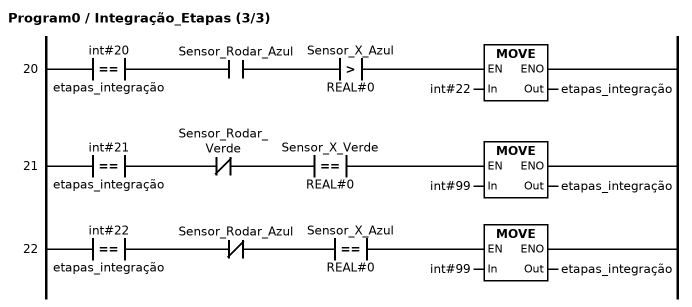
(* [picture p48: Program0 / Integração_Etapas, rungs 20-22] *)
(* Rung 20 *)
IF (int#20 = etapas_integração) AND Sensor_Rodar_Azul AND (Sensor_X_Azul > REAL#0) THEN
    etapas_integração := int#22;
END_IF;
(* Rung 21 *)
IF (int#21 = etapas_integração) AND NOT Sensor_Rodar_Verde AND (Sensor_X_Verde = REAL#0) THEN
    etapas_integração := int#99;
END_IF;
(* Rung 22 *)
IF (int#22 = etapas_integração) AND NOT Sensor_Rodar_Azul AND (Sensor_X_Azul = REAL#0) THEN
    etapas_integração := int#99;
END_IF;

(* Section Integração_Saídas: ladder, written here as Structured Text *)

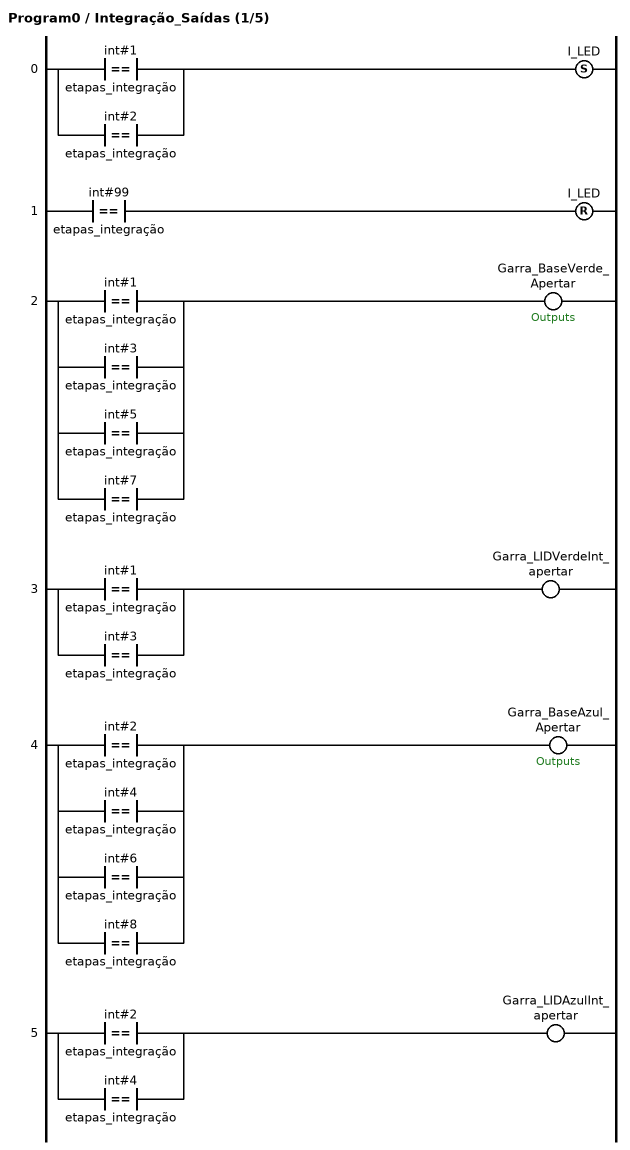
(* Rung 0 *)
IF (int#1 = etapas_integração) OR (int#2 = etapas_integração) THEN I_LED := TRUE; END_IF;
(* Rung 1 *)
IF int#99 = etapas_integração THEN I_LED := FALSE; END_IF;
(* Rung 2 *)
Garra_BaseVerde_Apertar := (int#1 = etapas_integração) OR (int#3 = etapas_integração) OR (int#5 = etapas_integração) OR (int#7 = etapas_integração);
(* Rung 3 *)
Garra_LIDVerdeInt_apertar := (int#1 = etapas_integração) OR (int#3 = etapas_integração);
(* Rung 4 *)
Garra_BaseAzul_Apertar := (int#2 = etapas_integração) OR (int#4 = etapas_integração) OR (int#6 = etapas_integração) OR (int#8 = etapas_integração);
(* Rung 5 *)
Garra_LIDAzulInt_apertar := (int#2 = etapas_integração) OR (int#4 = etapas_integração);

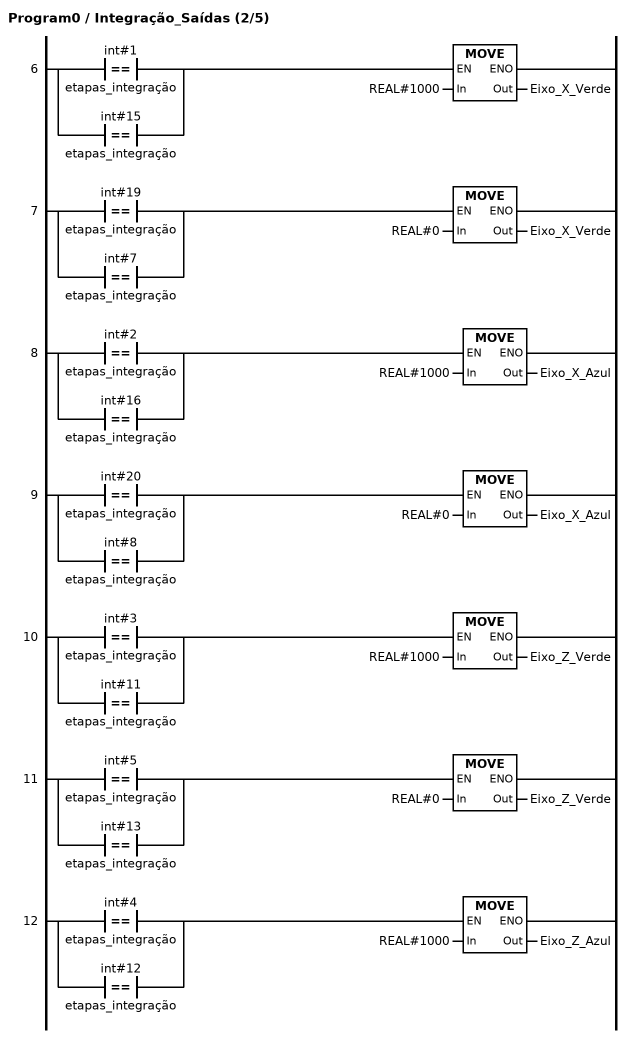
(* Rung 6 *)
IF (int#1 = etapas_integração) OR (int#15 = etapas_integração) THEN Eixo_X_Verde := REAL#1000; END_IF;
(* Rung 7 *)
IF (int#19 = etapas_integração) OR (int#7 = etapas_integração) THEN Eixo_X_Verde := REAL#0; END_IF;
(* Rung 8 *)
IF (int#2 = etapas_integração) OR (int#16 = etapas_integração) THEN Eixo_X_Azul := REAL#1000; END_IF;
(* Rung 9 *)
IF (int#20 = etapas_integração) OR (int#8 = etapas_integração) THEN Eixo_X_Azul := REAL#0; END_IF;
(* Rung 10 *)
IF (int#3 = etapas_integração) OR (int#11 = etapas_integração) THEN Eixo_Z_Verde := REAL#1000; END_IF;
(* Rung 11 *)
IF (int#5 = etapas_integração) OR (int#13 = etapas_integração) THEN Eixo_Z_Verde := REAL#0; END_IF;
(* Rung 12 *)
IF (int#4 = etapas_integração) OR (int#12 = etapas_integração) THEN Eixo_Z_Azul := REAL#1000; END_IF;

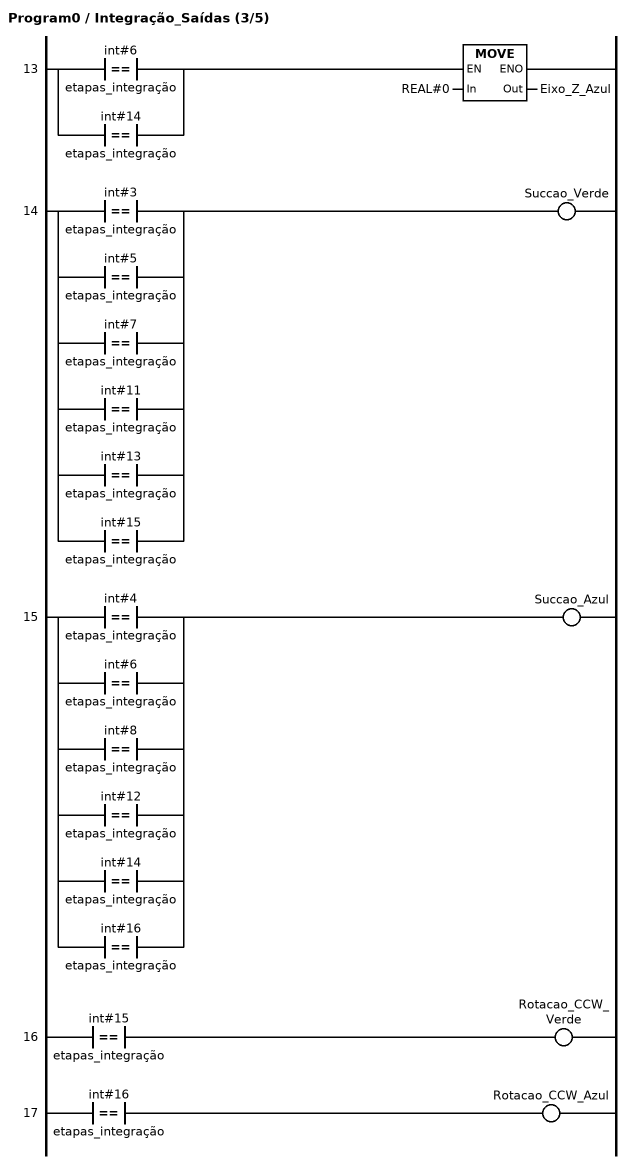
(* Rung 13 *)
IF (int#6 = etapas_integração) OR (int#14 = etapas_integração) THEN Eixo_Z_Azul := REAL#0; END_IF;
(* Rung 14 *)
Succao_Verde := (int#3 = etapas_integração) OR (int#5 = etapas_integração) OR (int#7 = etapas_integração) OR (int#11 = etapas_integração) OR (int#13 = etapas_integração) OR (int#15 = etapas_integração);
(* Rung 15 *)
Succao_Azul := (int#4 = etapas_integração) OR (int#6 = etapas_integração) OR (int#8 = etapas_integração) OR (int#12 = etapas_integração) OR (int#14 = etapas_integração) OR (int#16 = etapas_integração);
(* Rung 16 *)
Rotacao_CCW_Verde := int#15 = etapas_integração;
(* Rung 17 *)
Rotacao_CCW_Azul := int#16 = etapas_integração;

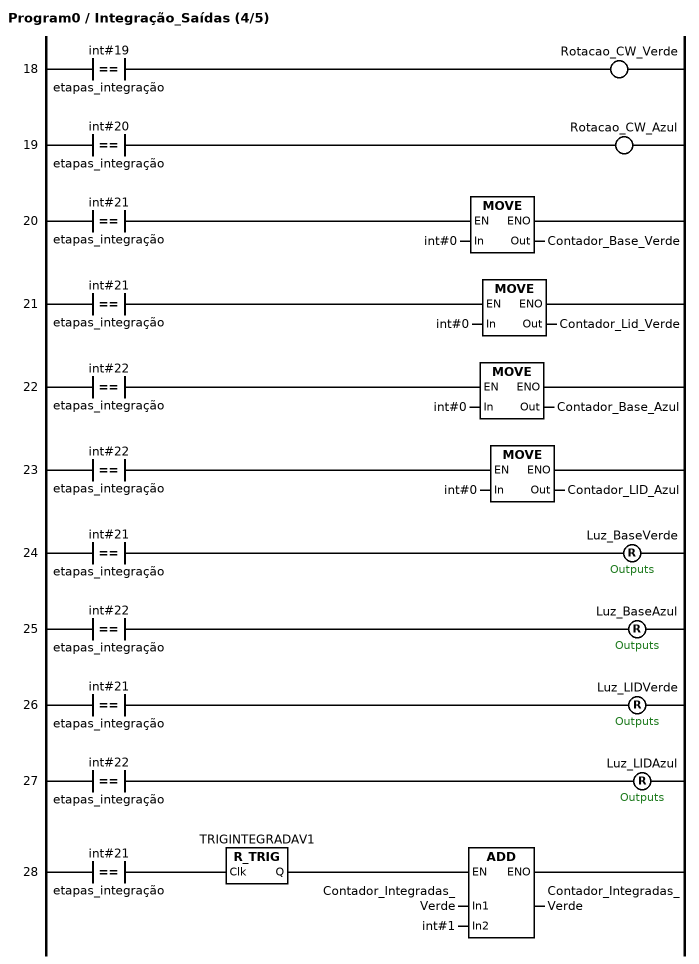
(* Rung 18 *)
Rotacao_CW_Verde := int#19 = etapas_integração;
(* Rung 19 *)
Rotacao_CW_Azul := int#20 = etapas_integração;
(* Rung 20 *)
IF int#21 = etapas_integração THEN Contador_Base_Verde := int#0; END_IF;
(* Rung 21 *)
IF int#21 = etapas_integração THEN Contador_Lid_Verde := int#0; END_IF;
(* Rung 22 *)
IF int#22 = etapas_integração THEN Contador_Base_Azul := int#0; END_IF;
(* Rung 23 *)
IF int#22 = etapas_integração THEN Contador_LID_Azul := int#0; END_IF;
(* Rung 24 *)
IF int#21 = etapas_integração THEN Luz_BaseVerde := FALSE; END_IF;
(* Rung 25 *)
IF int#22 = etapas_integração THEN Luz_BaseAzul := FALSE; END_IF;
(* Rung 26 *)
IF int#21 = etapas_integração THEN Luz_LIDVerde := FALSE; END_IF;
(* Rung 27 *)
IF int#22 = etapas_integração THEN Luz_LIDAzul := FALSE; END_IF;
(* Rung 28 *)
TRIGINTEGRADAV1(Clk := int#21 = etapas_integração);
IF TRIGINTEGRADAV1.Q THEN Contador_Integradas_Verde := Contador_Integradas_Verde + int#1; END_IF;

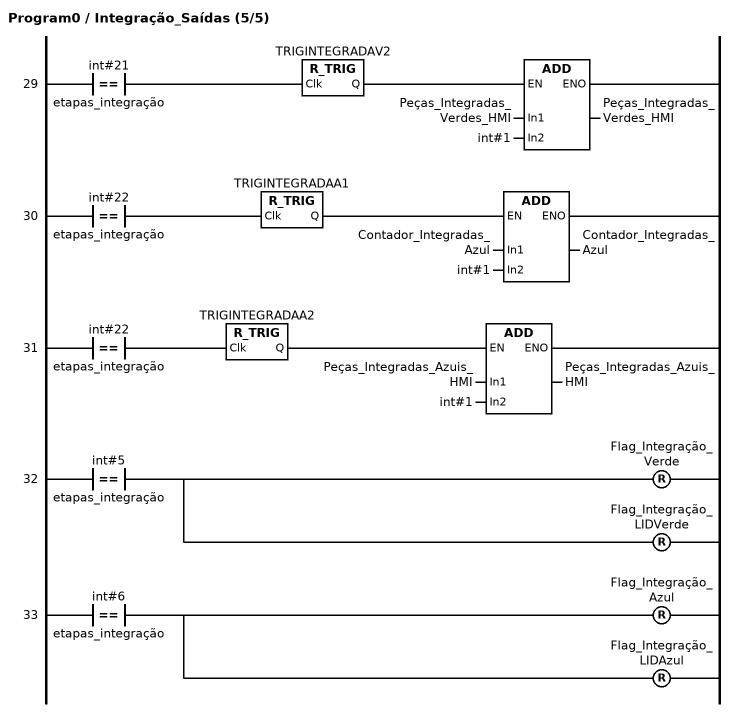
(* Rung 29 *)
TRIGINTEGRADAV2(Clk := int#21 = etapas_integração);
IF TRIGINTEGRADAV2.Q THEN Peças_Integradas_Verdes_HMI := Peças_Integradas_Verdes_HMI + int#1; END_IF;
(* Rung 30 *)
TRIGINTEGRADAA1(Clk := int#22 = etapas_integração);
IF TRIGINTEGRADAA1.Q THEN Contador_Integradas_Azul := Contador_Integradas_Azul + int#1; END_IF;
(* Rung 31 *)
TRIGINTEGRADAA2(Clk := int#22 = etapas_integração);
IF TRIGINTEGRADAA2.Q THEN Peças_Integradas_Azuis_HMI := Peças_Integradas_Azuis_HMI + int#1; END_IF;
(* Rung 32 *)
IF int#5 = etapas_integração THEN
    Flag_Integração_Verde := FALSE;
    Flag_Integração_LIDVerde := FALSE;
END_IF;
(* Rung 33 *)
IF int#6 = etapas_integração THEN
    Flag_Integração_Azul := FALSE;
    Flag_Integração_LIDAzul := FALSE;
END_IF;

(* Section Organização_Etapas: ladder, written here as Structured Text *)

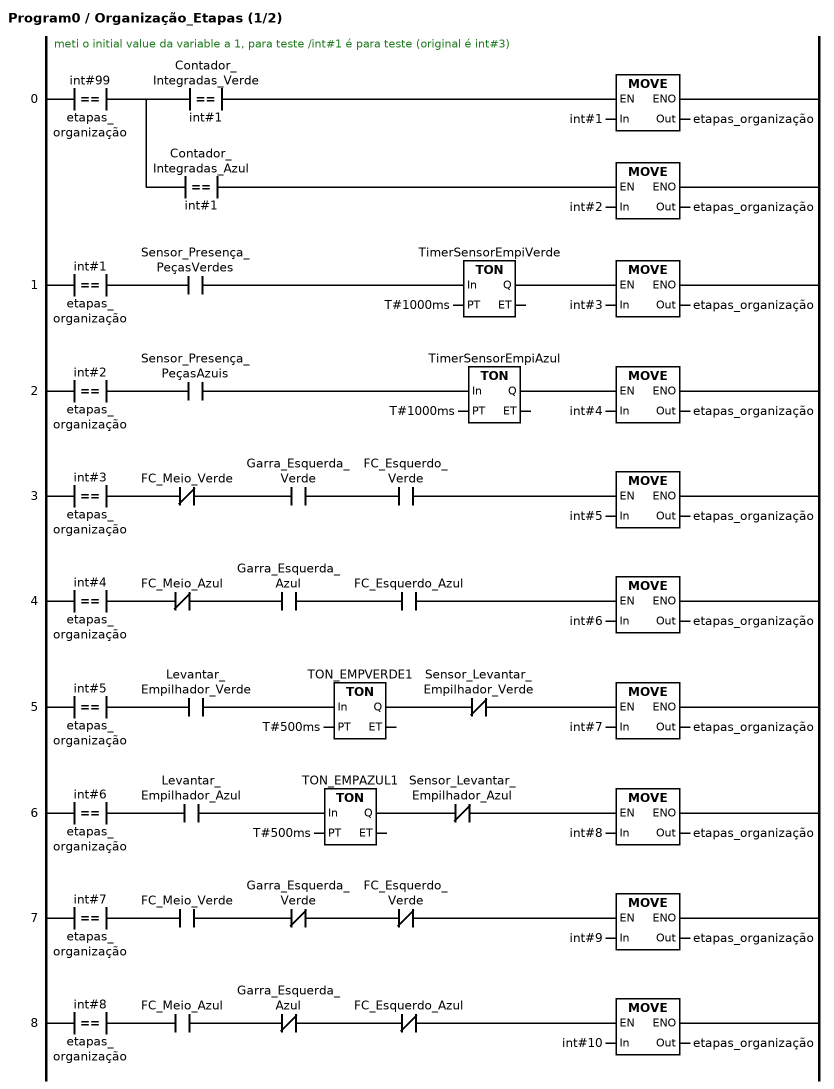
(* Rung 0: meti o initial value da variable a 1, para teste /int#1 é para teste (original é int#3) *)
_p11 := int#99 = etapas_organização;
IF (int#99 = etapas_organização) AND (Contador_Integradas_Verde = int#1) THEN
    etapas_organização := int#1;
END_IF;
IF _p11 AND (Contador_Integradas_Azul = int#1) THEN etapas_organização := int#2; END_IF;
(* Rung 1 *)
TimerSensorEmpiVerde(In := (int#1 = etapas_organização) AND Sensor_Presença_PeçasVerdes, PT := T#1000ms);
IF TimerSensorEmpiVerde.Q THEN etapas_organização := int#3; END_IF;
(* Rung 2 *)
TimerSensorEmpiAzul(In := (int#2 = etapas_organização) AND Sensor_Presença_PeçasAzuis, PT := T#1000ms);
IF TimerSensorEmpiAzul.Q THEN etapas_organização := int#4; END_IF;
(* Rung 3 *)
IF (int#3 = etapas_organização) AND NOT FC_Meio_Verde AND Garra_Esquerda_Verde AND FC_Esquerdo_Verde THEN
    etapas_organização := int#5;
END_IF;
(* Rung 4 *)
IF (int#4 = etapas_organização) AND NOT FC_Meio_Azul AND Garra_Esquerda_Azul AND FC_Esquerdo_Azul THEN
    etapas_organização := int#6;
END_IF;
(* Rung 5 *)
TON_EMPVERDE1(In := (int#5 = etapas_organização) AND Levantar_Empilhador_Verde, PT := T#500ms);
IF TON_EMPVERDE1.Q AND NOT Sensor_Levantar_Empilhador_Verde THEN etapas_organização := int#7; END_IF;
(* Rung 6 *)
TON_EMPAZUL1(In := (int#6 = etapas_organização) AND Levantar_Empilhador_Azul, PT := T#500ms);
IF TON_EMPAZUL1.Q AND NOT Sensor_Levantar_Empilhador_Azul THEN etapas_organização := int#8; END_IF;
(* Rung 7 *)
IF (int#7 = etapas_organização) AND FC_Meio_Verde AND NOT Garra_Esquerda_Verde AND NOT FC_Esquerdo_Verde THEN
    etapas_organização := int#9;
END_IF;
(* Rung 8 *)
IF (int#8 = etapas_organização) AND FC_Meio_Azul AND NOT Garra_Esquerda_Azul AND NOT FC_Esquerdo_Azul THEN
    etapas_organização := int#10;
END_IF;

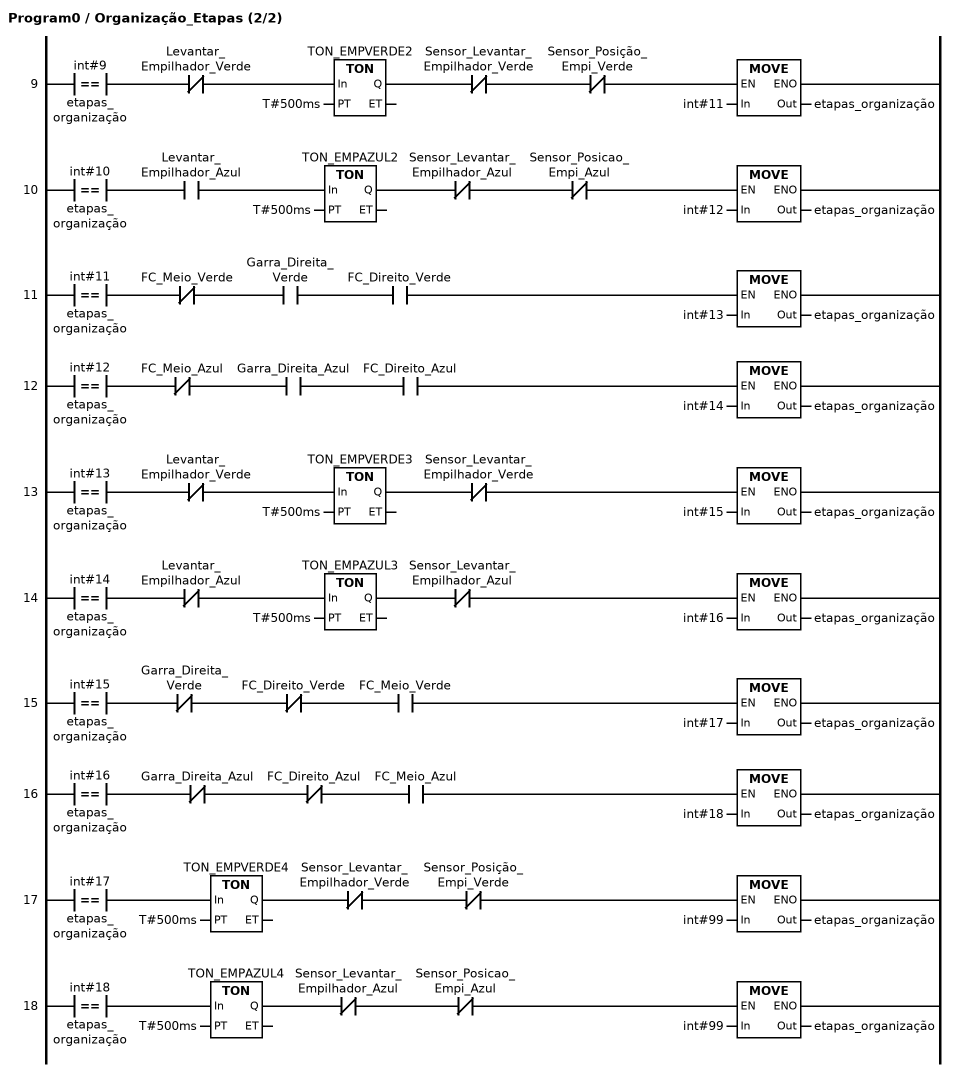
(* Rung 9 *)
TON_EMPVERDE2(In := (int#9 = etapas_organização) AND NOT Levantar_Empilhador_Verde, PT := T#500ms);
IF TON_EMPVERDE2.Q AND NOT Sensor_Levantar_Empilhador_Verde AND NOT Sensor_Posição_Empi_Verde THEN
    etapas_organização := int#11;
END_IF;
(* Rung 10 *)
TON_EMPAZUL2(In := (int#10 = etapas_organização) AND Levantar_Empilhador_Azul, PT := T#500ms);
IF TON_EMPAZUL2.Q AND NOT Sensor_Levantar_Empilhador_Azul AND NOT Sensor_Posicao_Empi_Azul THEN
    etapas_organização := int#12;
END_IF;
(* Rung 11 *)
IF (int#11 = etapas_organização) AND NOT FC_Meio_Verde AND Garra_Direita_Verde AND FC_Direito_Verde THEN
    etapas_organização := int#13;
END_IF;
(* Rung 12 *)
IF (int#12 = etapas_organização) AND NOT FC_Meio_Azul AND Garra_Direita_Azul AND FC_Direito_Azul THEN
    etapas_organização := int#14;
END_IF;
(* Rung 13 *)
TON_EMPVERDE3(In := (int#13 = etapas_organização) AND NOT Levantar_Empilhador_Verde, PT := T#500ms);
IF TON_EMPVERDE3.Q AND NOT Sensor_Levantar_Empilhador_Verde THEN etapas_organização := int#15; END_IF;
(* Rung 14 *)
TON_EMPAZUL3(In := (int#14 = etapas_organização) AND NOT Levantar_Empilhador_Azul, PT := T#500ms);
IF TON_EMPAZUL3.Q AND NOT Sensor_Levantar_Empilhador_Azul THEN etapas_organização := int#16; END_IF;
(* Rung 15 *)
IF (int#15 = etapas_organização) AND NOT Garra_Direita_Verde AND NOT FC_Direito_Verde AND FC_Meio_Verde THEN
    etapas_organização := int#17;
END_IF;
(* Rung 16 *)
IF (int#16 = etapas_organização) AND NOT Garra_Direita_Azul AND NOT FC_Direito_Azul AND FC_Meio_Azul THEN
    etapas_organização := int#18;
END_IF;
(* Rung 17 *)
TON_EMPVERDE4(In := int#17 = etapas_organização, PT := T#500ms);
IF TON_EMPVERDE4.Q AND NOT Sensor_Levantar_Empilhador_Verde AND NOT Sensor_Posição_Empi_Verde THEN
    etapas_organização := int#99;
END_IF;
(* Rung 18 *)
TON_EMPAZUL4(In := int#18 = etapas_organização, PT := T#500ms);
IF TON_EMPAZUL4.Q AND NOT Sensor_Levantar_Empilhador_Azul AND NOT Sensor_Posicao_Empi_Azul THEN
    etapas_organização := int#99;
END_IF;

(* Section Organização_Saídas: ladder, written here as Structured Text *)

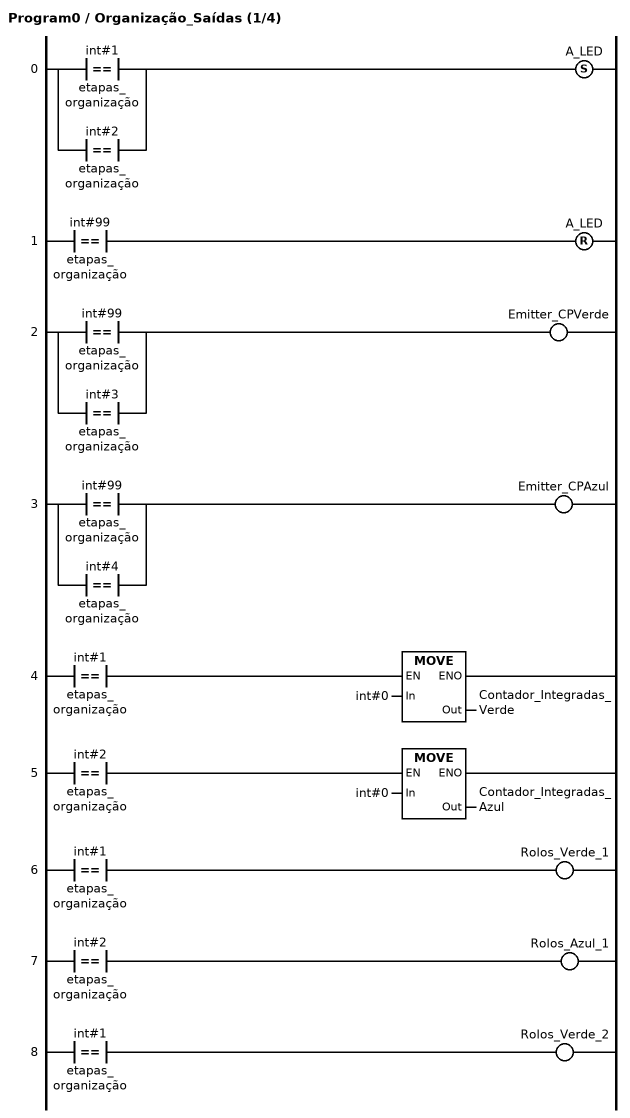
(* Rung 0 *)
IF (int#1 = etapas_organização) OR (int#2 = etapas_organização) THEN A_LED := TRUE; END_IF;
(* Rung 1 *)
IF int#99 = etapas_organização THEN A_LED := FALSE; END_IF;
(* Rung 2 *)
Emitter_CPVerde := (int#99 = etapas_organização) OR (int#3 = etapas_organização);
(* Rung 3 *)
Emitter_CPAzul := (int#99 = etapas_organização) OR (int#4 = etapas_organização);
(* Rung 4 *)
IF int#1 = etapas_organização THEN Contador_Integradas_Verde := int#0; END_IF;
(* Rung 5 *)
IF int#2 = etapas_organização THEN Contador_Integradas_Azul := int#0; END_IF;
(* Rung 6 *)
Rolos_Verde_1 := int#1 = etapas_organização;
(* Rung 7 *)
Rolos_Azul_1 := int#2 = etapas_organização;
(* Rung 8 *)
Rolos_Verde_2 := int#1 = etapas_organização;

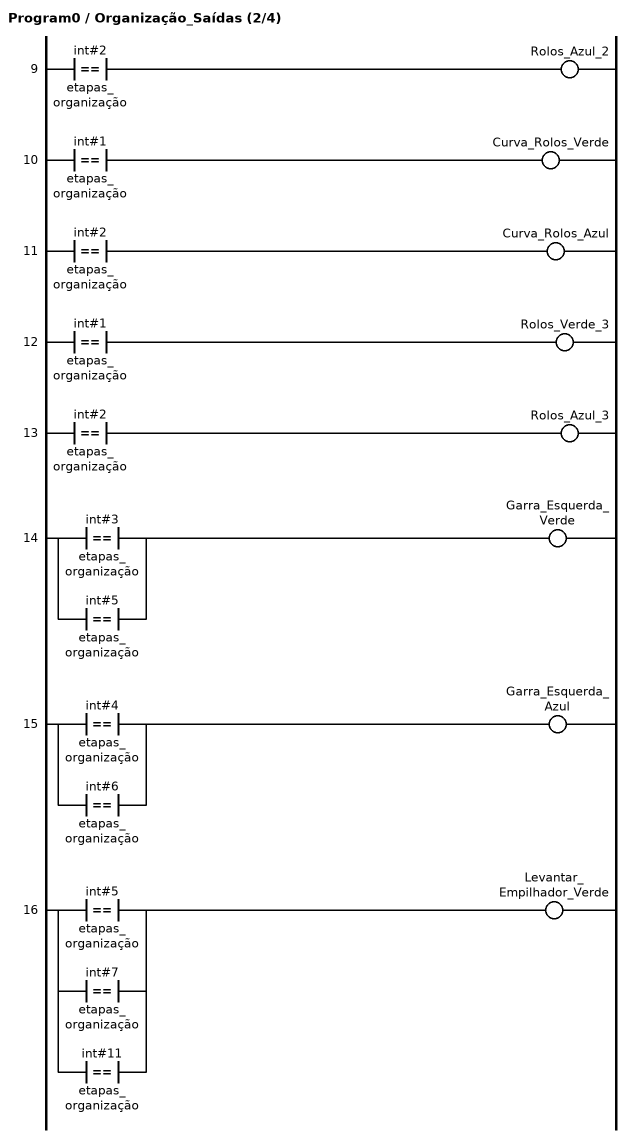
(* Rung 9 *)
Rolos_Azul_2 := int#2 = etapas_organização;
(* Rung 10 *)
Curva_Rolos_Verde := int#1 = etapas_organização;
(* Rung 11 *)
Curva_Rolos_Azul := int#2 = etapas_organização;
(* Rung 12 *)
Rolos_Verde_3 := int#1 = etapas_organização;
(* Rung 13 *)
Rolos_Azul_3 := int#2 = etapas_organização;
(* Rung 14 *)
Garra_Esquerda_Verde := (int#3 = etapas_organização) OR (int#5 = etapas_organização);
(* Rung 15 *)
Garra_Esquerda_Azul := (int#4 = etapas_organização) OR (int#6 = etapas_organização);
(* Rung 16 *)
Levantar_Empilhador_Verde := (int#5 = etapas_organização) OR (int#7 = etapas_organização) OR (int#11 = etapas_organização);

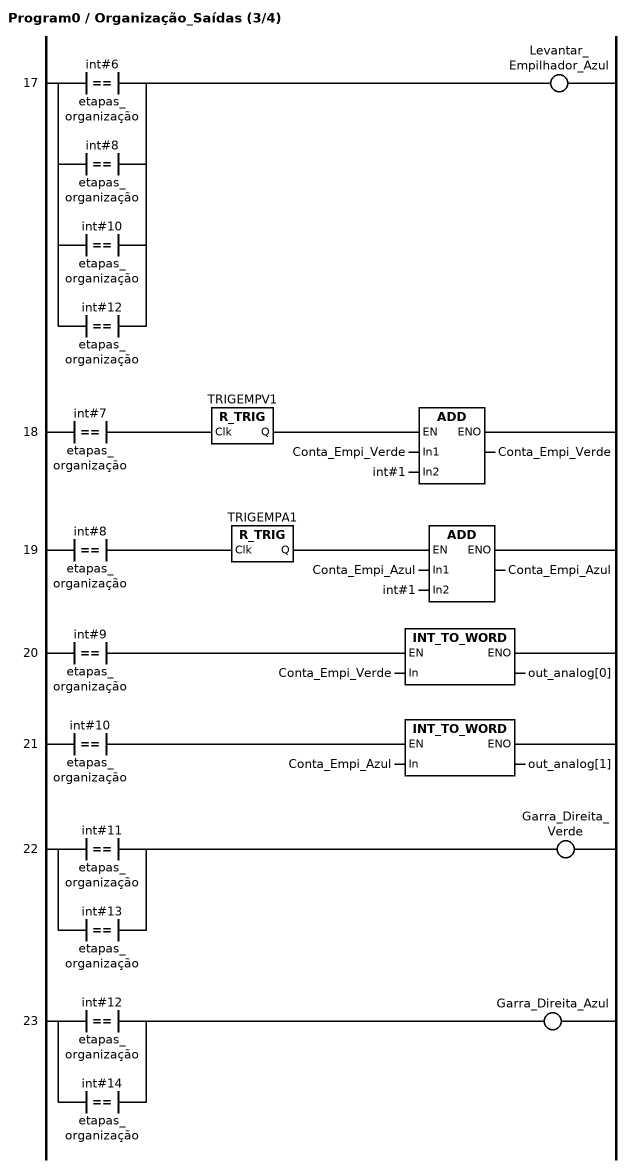
(* Rung 17 *)
Levantar_Empilhador_Azul := (int#6 = etapas_organização) OR (int#8 = etapas_organização) OR (int#10 = etapas_organização) OR (int#12 = etapas_organização);
(* Rung 18 *)
TRIGEMPV1(Clk := int#7 = etapas_organização);
IF TRIGEMPV1.Q THEN Conta_Empi_Verde := Conta_Empi_Verde + int#1; END_IF;
(* Rung 19 *)
TRIGEMPA1(Clk := int#8 = etapas_organização);
IF TRIGEMPA1.Q THEN Conta_Empi_Azul := Conta_Empi_Azul + int#1; END_IF;
(* Rung 20 *)
IF int#9 = etapas_organização THEN out_analog[0] := INT_TO_WORD(In := Conta_Empi_Verde); END_IF;
(* Rung 21 *)
IF int#10 = etapas_organização THEN out_analog[1] := INT_TO_WORD(In := Conta_Empi_Azul); END_IF;
(* Rung 22 *)
Garra_Direita_Verde := (int#11 = etapas_organização) OR (int#13 = etapas_organização);
(* Rung 23 *)
Garra_Direita_Azul := (int#12 = etapas_organização) OR (int#14 = etapas_organização);

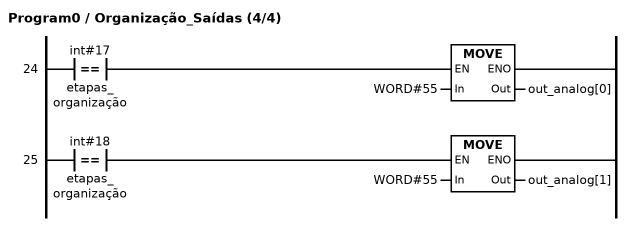
(* Rung 24 *)
IF int#17 = etapas_organização THEN out_analog[0] := WORD#55; END_IF;
(* Rung 25 *)
IF int#18 = etapas_organização THEN out_analog[1] := WORD#55; END_IF;

(* Section ExpediçãoVerde_Etapas: ladder, written here as Structured Text *)

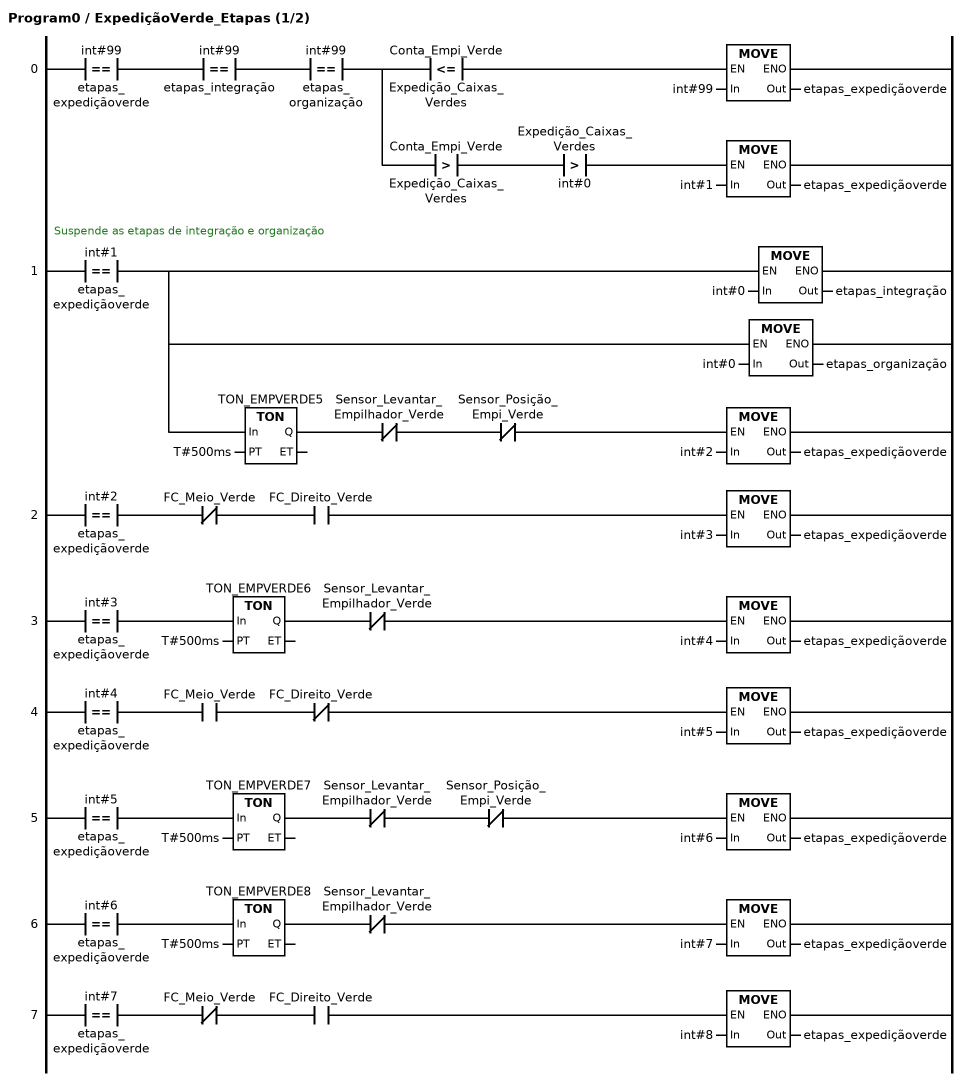
(* Rung 0 *)
_p12 := (int#99 = etapas_expediçãoverde) AND (int#99 = etapas_integração) AND (int#99 = etapas_organização);
IF _p12 AND (Conta_Empi_Verde <= Expedição_Caixas_Verdes) THEN etapas_expediçãoverde := int#99; END_IF;
IF _p12 AND (Conta_Empi_Verde > Expedição_Caixas_Verdes) AND (Expedição_Caixas_Verdes > int#0) THEN
    etapas_expediçãoverde := int#1;
END_IF;
(* Rung 1: Suspende as etapas de integração e organização *)
IF int#1 = etapas_expediçãoverde THEN
    etapas_integração := int#0;
    etapas_organização := int#0;
END_IF;
TON_EMPVERDE5(In := int#1 = etapas_expediçãoverde, PT := T#500ms);
IF TON_EMPVERDE5.Q AND NOT Sensor_Levantar_Empilhador_Verde AND NOT Sensor_Posição_Empi_Verde THEN
    etapas_expediçãoverde := int#2;
END_IF;
(* Rung 2 *)
IF (int#2 = etapas_expediçãoverde) AND NOT FC_Meio_Verde AND FC_Direito_Verde THEN
    etapas_expediçãoverde := int#3;
END_IF;
(* Rung 3 *)
TON_EMPVERDE6(In := int#3 = etapas_expediçãoverde, PT := T#500ms);
IF TON_EMPVERDE6.Q AND NOT Sensor_Levantar_Empilhador_Verde THEN etapas_expediçãoverde := int#4; END_IF;
(* Rung 4 *)
IF (int#4 = etapas_expediçãoverde) AND FC_Meio_Verde AND NOT FC_Direito_Verde THEN
    etapas_expediçãoverde := int#5;
END_IF;
(* Rung 5 *)
TON_EMPVERDE7(In := int#5 = etapas_expediçãoverde, PT := T#500ms);
IF TON_EMPVERDE7.Q AND NOT Sensor_Levantar_Empilhador_Verde AND NOT Sensor_Posição_Empi_Verde THEN
    etapas_expediçãoverde := int#6;
END_IF;
(* Rung 6 *)
TON_EMPVERDE8(In := int#6 = etapas_expediçãoverde, PT := T#500ms);
IF TON_EMPVERDE8.Q AND NOT Sensor_Levantar_Empilhador_Verde THEN etapas_expediçãoverde := int#7; END_IF;
(* Rung 7 *)
IF (int#7 = etapas_expediçãoverde) AND NOT FC_Meio_Verde AND FC_Direito_Verde THEN
    etapas_expediçãoverde := int#8;
END_IF;

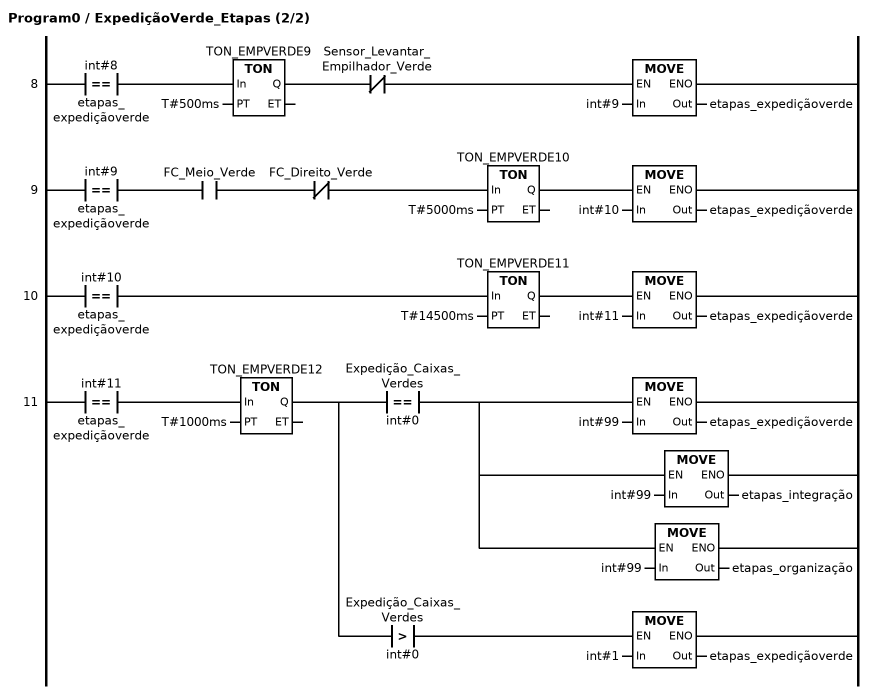
(* Rung 8 *)
TON_EMPVERDE9(In := int#8 = etapas_expediçãoverde, PT := T#500ms);
IF TON_EMPVERDE9.Q AND NOT Sensor_Levantar_Empilhador_Verde THEN etapas_expediçãoverde := int#9; END_IF;
(* Rung 9 *)
TON_EMPVERDE10(In := (int#9 = etapas_expediçãoverde) AND FC_Meio_Verde AND NOT FC_Direito_Verde, PT := T#5000ms);
IF TON_EMPVERDE10.Q THEN etapas_expediçãoverde := int#10; END_IF;
(* Rung 10 *)
TON_EMPVERDE11(In := int#10 = etapas_expediçãoverde, PT := T#14500ms);
IF TON_EMPVERDE11.Q THEN etapas_expediçãoverde := int#11; END_IF;
(* Rung 11 *)
TON_EMPVERDE12(In := int#11 = etapas_expediçãoverde, PT := T#1000ms);
_p13 := TON_EMPVERDE12.Q AND (Expedição_Caixas_Verdes = int#0);
IF _p13 THEN
    etapas_expediçãoverde := int#99;
    etapas_integração := int#99;
    etapas_organização := int#99;
END_IF;
IF TON_EMPVERDE12.Q AND (Expedição_Caixas_Verdes > int#0) THEN etapas_expediçãoverde := int#1; END_IF;

(* Section ExpediçãoVerde_Saídas: ladder, written here as Structured Text *)

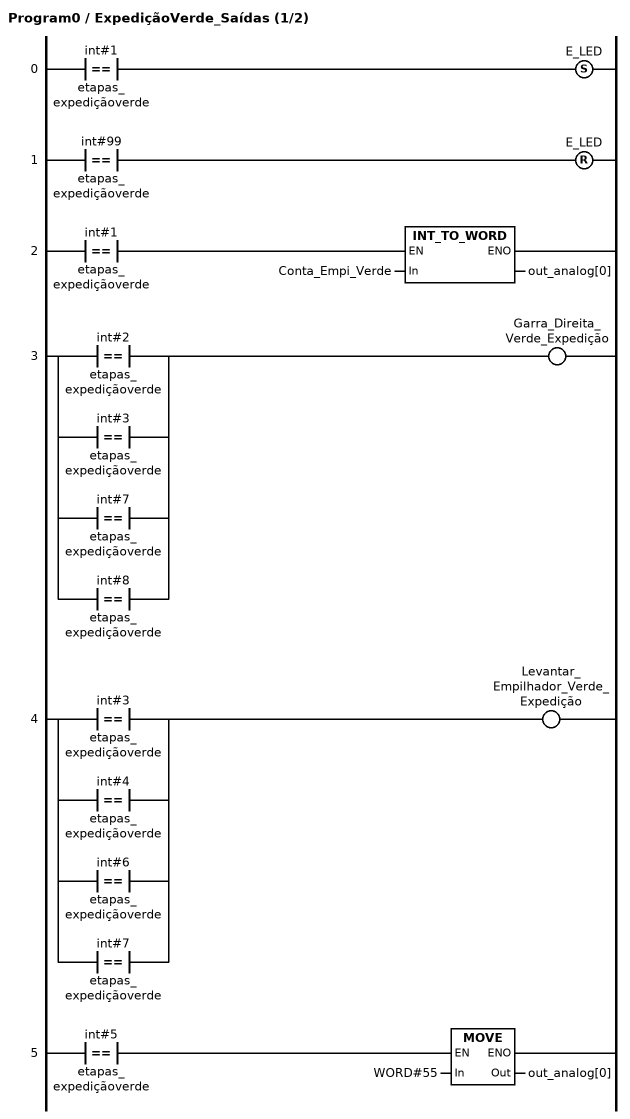
(* Rung 0 *)
IF int#1 = etapas_expediçãoverde THEN E_LED := TRUE; END_IF;
(* Rung 1 *)
IF int#99 = etapas_expediçãoverde THEN E_LED := FALSE; END_IF;
(* Rung 2 *)
IF int#1 = etapas_expediçãoverde THEN out_analog[0] := INT_TO_WORD(In := Conta_Empi_Verde); END_IF;
(* Rung 3 *)
Garra_Direita_Verde_Expedição := (int#2 = etapas_expediçãoverde) OR (int#3 = etapas_expediçãoverde) OR (int#7 = etapas_expediçãoverde) OR (int#8 = etapas_expediçãoverde);
(* Rung 4 *)
Levantar_Empilhador_Verde_Expedição := (int#3 = etapas_expediçãoverde) OR (int#4 = etapas_expediçãoverde) OR (int#6 = etapas_expediçãoverde) OR (int#7 = etapas_expediçãoverde);
(* Rung 5 *)
IF int#5 = etapas_expediçãoverde THEN out_analog[0] := WORD#55; END_IF;

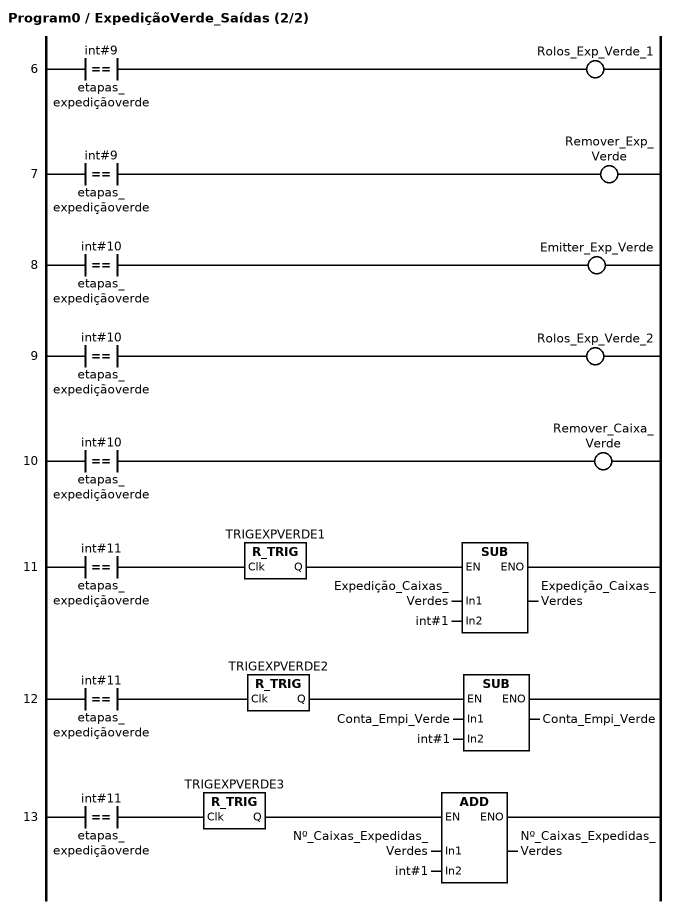
(* Rung 6 *)
Rolos_Exp_Verde_1 := int#9 = etapas_expediçãoverde;
(* Rung 7 *)
Remover_Exp_Verde := int#9 = etapas_expediçãoverde;
(* Rung 8 *)
Emitter_Exp_Verde := int#10 = etapas_expediçãoverde;
(* Rung 9 *)
Rolos_Exp_Verde_2 := int#10 = etapas_expediçãoverde;
(* Rung 10 *)
Remover_Caixa_Verde := int#10 = etapas_expediçãoverde;
(* Rung 11 *)
TRIGEXPVERDE1(Clk := int#11 = etapas_expediçãoverde);
IF TRIGEXPVERDE1.Q THEN Expedição_Caixas_Verdes := Expedição_Caixas_Verdes - int#1; END_IF;
(* Rung 12 *)
TRIGEXPVERDE2(Clk := int#11 = etapas_expediçãoverde);
IF TRIGEXPVERDE2.Q THEN Conta_Empi_Verde := Conta_Empi_Verde - int#1; END_IF;
(* Rung 13 *)
TRIGEXPVERDE3(Clk := int#11 = etapas_expediçãoverde);
IF TRIGEXPVERDE3.Q THEN Nº_Caixas_Expedidas_Verdes := Nº_Caixas_Expedidas_Verdes + int#1; END_IF;

(* Section ExpediçãoAzul_Etapas: ladder, written here as Structured Text *)

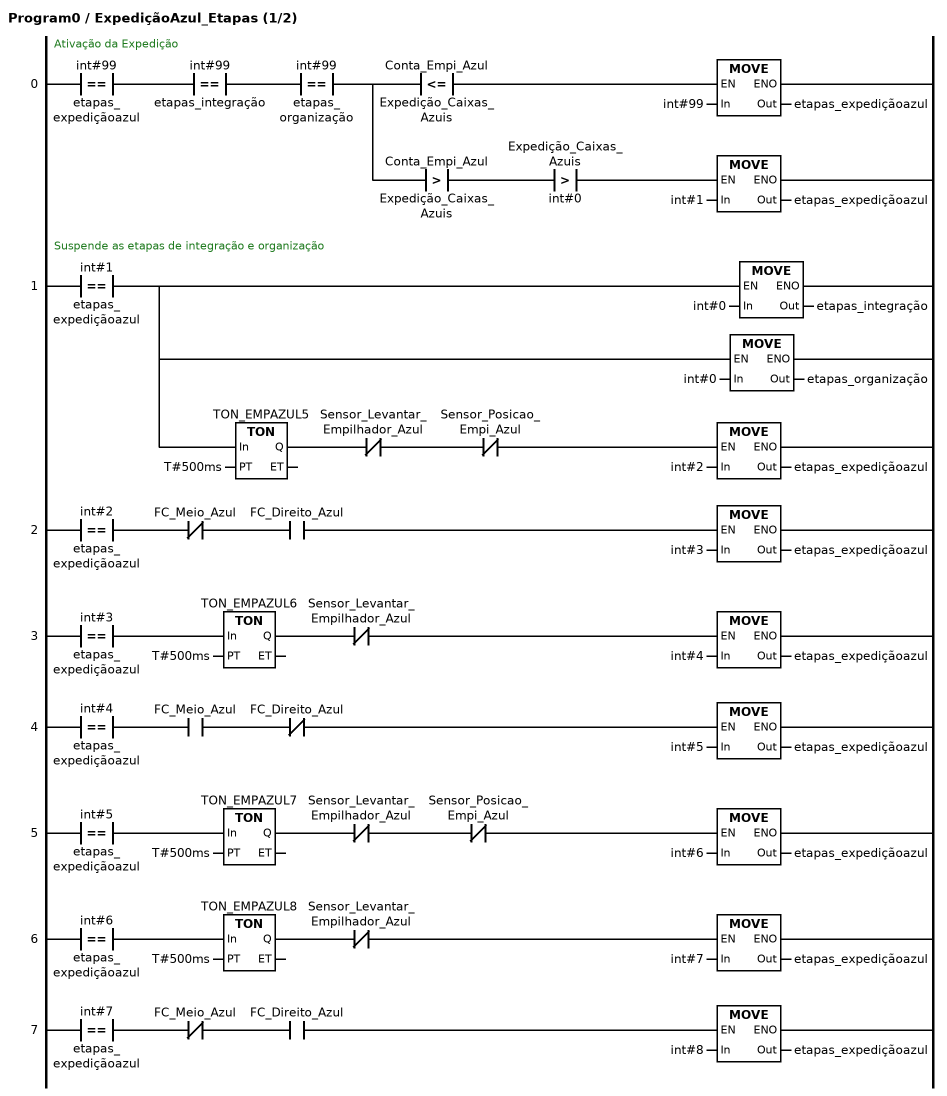
(* Rung 0: Ativação da Expedição *)
_p14 := (int#99 = etapas_expediçãoazul) AND (int#99 = etapas_integração) AND (int#99 = etapas_organização);
IF _p14 AND (Conta_Empi_Azul <= Expedição_Caixas_Azuis) THEN etapas_expediçãoazul := int#99; END_IF;
IF _p14 AND (Conta_Empi_Azul > Expedição_Caixas_Azuis) AND (Expedição_Caixas_Azuis > int#0) THEN
    etapas_expediçãoazul := int#1;
END_IF;
(* Rung 1: Suspende as etapas de integração e organização *)
IF int#1 = etapas_expediçãoazul THEN
    etapas_integração := int#0;
    etapas_organização := int#0;
END_IF;
TON_EMPAZUL5(In := int#1 = etapas_expediçãoazul, PT := T#500ms);
IF TON_EMPAZUL5.Q AND NOT Sensor_Levantar_Empilhador_Azul AND NOT Sensor_Posicao_Empi_Azul THEN
    etapas_expediçãoazul := int#2;
END_IF;
(* Rung 2 *)
IF (int#2 = etapas_expediçãoazul) AND NOT FC_Meio_Azul AND FC_Direito_Azul THEN
    etapas_expediçãoazul := int#3;
END_IF;
(* Rung 3 *)
TON_EMPAZUL6(In := int#3 = etapas_expediçãoazul, PT := T#500ms);
IF TON_EMPAZUL6.Q AND NOT Sensor_Levantar_Empilhador_Azul THEN etapas_expediçãoazul := int#4; END_IF;
(* Rung 4 *)
IF (int#4 = etapas_expediçãoazul) AND FC_Meio_Azul AND NOT FC_Direito_Azul THEN
    etapas_expediçãoazul := int#5;
END_IF;
(* Rung 5 *)
TON_EMPAZUL7(In := int#5 = etapas_expediçãoazul, PT := T#500ms);
IF TON_EMPAZUL7.Q AND NOT Sensor_Levantar_Empilhador_Azul AND NOT Sensor_Posicao_Empi_Azul THEN
    etapas_expediçãoazul := int#6;
END_IF;
(* Rung 6 *)
TON_EMPAZUL8(In := int#6 = etapas_expediçãoazul, PT := T#500ms);
IF TON_EMPAZUL8.Q AND NOT Sensor_Levantar_Empilhador_Azul THEN etapas_expediçãoazul := int#7; END_IF;
(* Rung 7 *)
IF (int#7 = etapas_expediçãoazul) AND NOT FC_Meio_Azul AND FC_Direito_Azul THEN
    etapas_expediçãoazul := int#8;
END_IF;

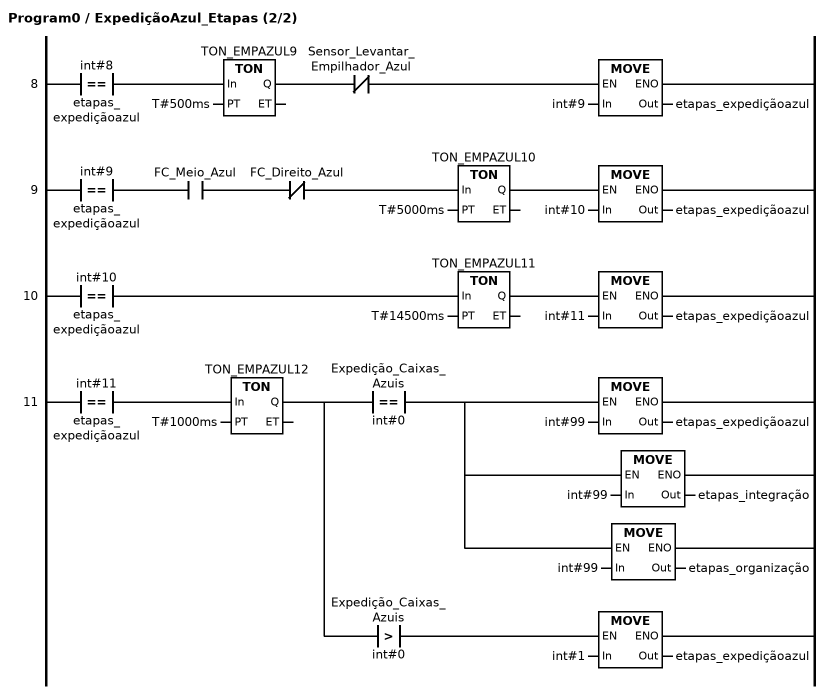
(* Rung 8 *)
TON_EMPAZUL9(In := int#8 = etapas_expediçãoazul, PT := T#500ms);
IF TON_EMPAZUL9.Q AND NOT Sensor_Levantar_Empilhador_Azul THEN etapas_expediçãoazul := int#9; END_IF;
(* Rung 9 *)
TON_EMPAZUL10(In := (int#9 = etapas_expediçãoazul) AND FC_Meio_Azul AND NOT FC_Direito_Azul, PT := T#5000ms);
IF TON_EMPAZUL10.Q THEN etapas_expediçãoazul := int#10; END_IF;
(* Rung 10 *)
TON_EMPAZUL11(In := int#10 = etapas_expediçãoazul, PT := T#14500ms);
IF TON_EMPAZUL11.Q THEN etapas_expediçãoazul := int#11; END_IF;
(* Rung 11 *)
TON_EMPAZUL12(In := int#11 = etapas_expediçãoazul, PT := T#1000ms);
_p15 := TON_EMPAZUL12.Q AND (Expedição_Caixas_Azuis = int#0);
IF _p15 THEN
    etapas_expediçãoazul := int#99;
    etapas_integração := int#99;
    etapas_organização := int#99;
END_IF;
IF TON_EMPAZUL12.Q AND (Expedição_Caixas_Azuis > int#0) THEN etapas_expediçãoazul := int#1; END_IF;

(* Section ExpediçãoAzul_Saídas: ladder, written here as Structured Text *)

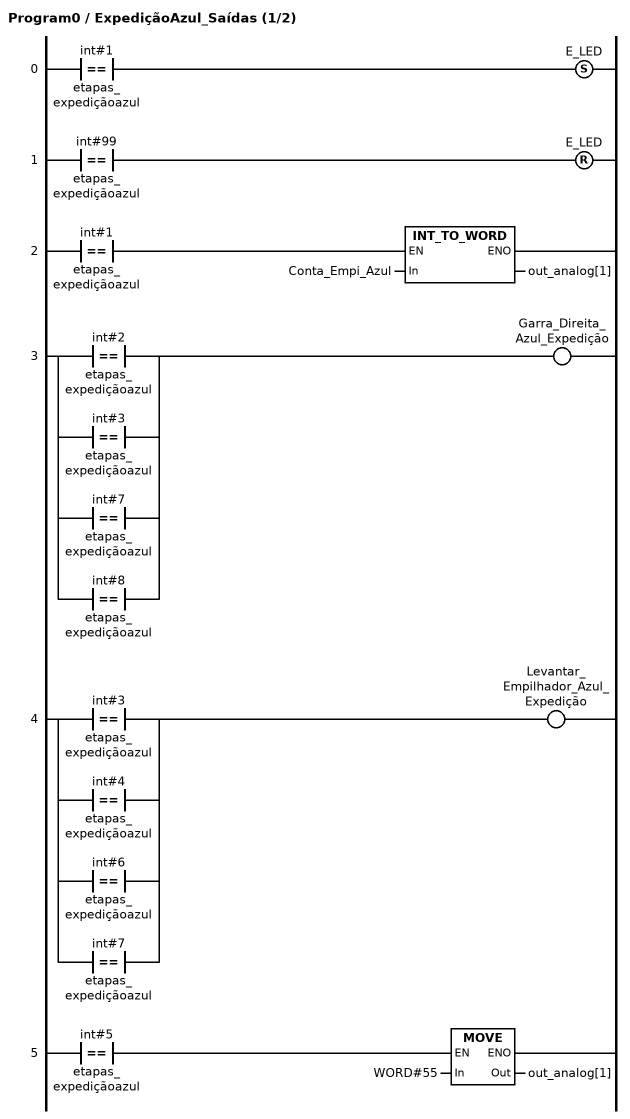
(* Rung 0 *)
IF int#1 = etapas_expediçãoazul THEN E_LED := TRUE; END_IF;
(* Rung 1 *)
IF int#99 = etapas_expediçãoazul THEN E_LED := FALSE; END_IF;
(* Rung 2 *)
IF int#1 = etapas_expediçãoazul THEN out_analog[1] := INT_TO_WORD(In := Conta_Empi_Azul); END_IF;
(* Rung 3 *)
Garra_Direita_Azul_Expedição := (int#2 = etapas_expediçãoazul) OR (int#3 = etapas_expediçãoazul) OR (int#7 = etapas_expediçãoazul) OR (int#8 = etapas_expediçãoazul);
(* Rung 4 *)
Levantar_Empilhador_Azul_Expedição := (int#3 = etapas_expediçãoazul) OR (int#4 = etapas_expediçãoazul) OR (int#6 = etapas_expediçãoazul) OR (int#7 = etapas_expediçãoazul);
(* Rung 5 *)
IF int#5 = etapas_expediçãoazul THEN out_analog[1] := WORD#55; END_IF;

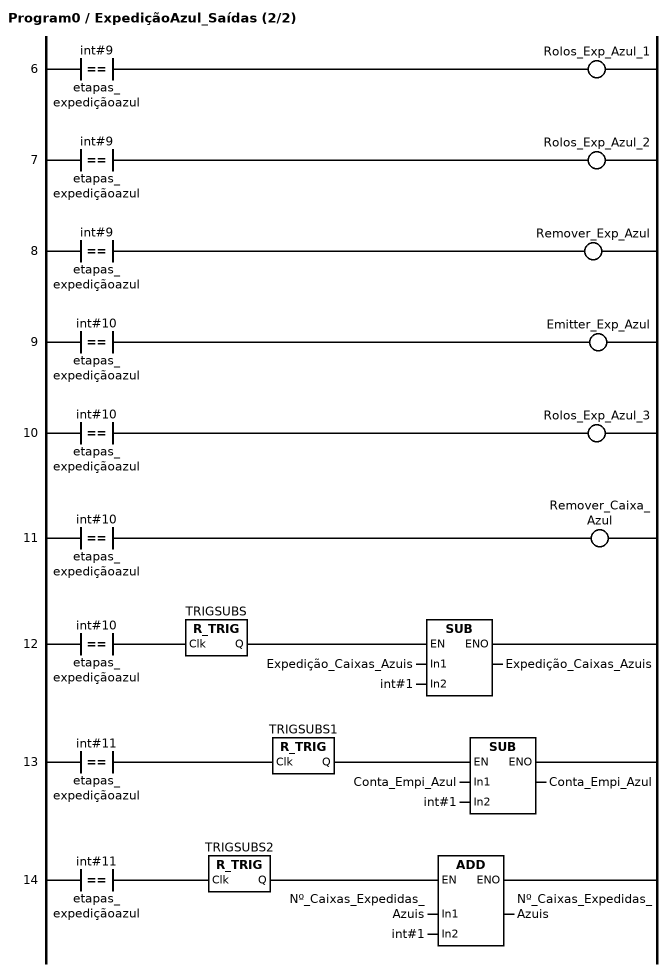
(* Rung 6 *)
Rolos_Exp_Azul_1 := int#9 = etapas_expediçãoazul;
(* Rung 7 *)
Rolos_Exp_Azul_2 := int#9 = etapas_expediçãoazul;
(* Rung 8 *)
Remover_Exp_Azul := int#9 = etapas_expediçãoazul;
(* Rung 9 *)
Emitter_Exp_Azul := int#10 = etapas_expediçãoazul;
(* Rung 10 *)
Rolos_Exp_Azul_3 := int#10 = etapas_expediçãoazul;
(* Rung 11 *)
Remover_Caixa_Azul := int#10 = etapas_expediçãoazul;
(* Rung 12 *)
TRIGSUBS(Clk := int#10 = etapas_expediçãoazul);
IF TRIGSUBS.Q THEN Expedição_Caixas_Azuis := Expedição_Caixas_Azuis - int#1; END_IF;
(* Rung 13 *)
TRIGSUBS1(Clk := int#11 = etapas_expediçãoazul);
IF TRIGSUBS1.Q THEN Conta_Empi_Azul := Conta_Empi_Azul - int#1; END_IF;
(* Rung 14 *)
TRIGSUBS2(Clk := int#11 = etapas_expediçãoazul);
IF TRIGSUBS2.Q THEN Nº_Caixas_Expedidas_Azuis := Nº_Caixas_Expedidas_Azuis + int#1; END_IF;
END_PROGRAM